var_global bInput    AT %I0.0 : bool; nAnalog   AT %I2    : int; bOutput   AT %Q0.0 : bool; nSetpoint AT %Q4   : dint; end_var

(* stored: Version 1.1.0.1, ProductVersion 3.1.4024.16
   GVL GVL_Syntax_Address: Id {c0f546e2-e66f-4137-95fc-87f0e029462f} *)
